//在PLC 重新启动的时候 关闭所以Socket
PROGRAM CloseAllSocket
VAR
	fbSocketCloseAll : FB_SocketCloseAll;
    bCloseAll        : BOOL := TRUE;
	tInit 			 : TON;
END_VAR

tInit(IN:=TRUE , PT:=T#10MS , Q=> , ET=> );
IF NOT tInit.Q THEN
	fbSocketCloseAll( bExecute:= FALSE );
	RETURN;
END_IF

IF bCloseAll THEN(*On PLC reset or program download close all old connections *)
    bCloseAll := FALSE;
	fbSocketCloseAll(
		sSrvNetId:= '', 
		bExecute:= TRUE, 
		tTimeout:= T#10S, 
		bBusy=> , 
		bError=> , 
		nErrId=> );
ELSE
    fbSocketCloseAll( bExecute:= FALSE );
END_IF

ACTION VersionLog:
(*
版本: V1.0.0.0
说明:
	1. 首个版本
//**************************************************//
版本: V1.0.0.1
说明:
	1. 上电后延时关闭所有旧的连接
//**************************************************//
*)
END_ACTION

END_PROGRAM

(* stored: Version 1.1.0.1, ProductVersion 3.1.4024.4
   POU CloseAllSocket: Id {7b565654-c153-4c7d-9f62-ba04530f34f6}, SpecialFunc None
   Action VersionLog: Id {000443c0-5947-4bc9-b5c7-42a04627e261} *)
